FUNCTION_BLOCK SOL_MDL (* Solenoid Model *)
  (* Standard: 61499-1; Classification: Simulation *)
  (* Version 0.1, 2005-06-01, JHC, Holobloc Inc, Recompiled with new emitter. *)
  (* Version 0.0, 2004-09-23, JHC, Rockwell Automation, Simplified, derived from CNV_MDL1. *)
  (* Compiler header: package fb.rt.mva; *)
  (* Compiler Java Sun JDK 1.4.2 *)
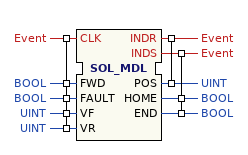
  EVENT_INPUT
    CLK WITH FWD, VF, FAULT, VR; (* Simulation Clock Event *)
  END_EVENT
  EVENT_OUTPUT
    INDR WITH POS; (* Change in Rendering Data *)
    INDS WITH HOME, END; (* Change in Sensor Data *)
  END_EVENT
  VAR_INPUT
    FWD : BOOL; (* Forward motion command *)
    FAULT : BOOL; (* Fault Condition *)
    VF : UINT := 50; (* Forward Speed in % per CLK event *)
    VR : UINT := 50; (* Retract Speed in % per CLK event *)
  END_VAR
  VAR_OUTPUT
    POS : UINT; (* Solenoid Position in % of Conveyor Length *)
    HOME : BOOL; (* Solenoid Fully Retracted *)
    END : BOOL; (* Solenoid Fully Advanced *)
  END_VAR
  ALGORITHM CLK IN Java:
if(FAULT.value) return;
if(FWD.value){
   if(END.value) return;
   if(HOME.value){
      HOME.value = false;
      INDS.serviceEvent(this);}
   POS.value += VF.value;
   if(POS.value >= 100){
      POS.value=100;
      END.value=true;
      INDS.serviceEvent(this);}}
else{
   if (HOME.value) return;
   if(END.value){
      END.value = false;
      INDS.serviceEvent(this);}
   POS.value -= VR.value;
   if(POS.value <= 0){
      POS.value=0;
      HOME.value=true;
      INDS.serviceEvent(this);}}
INDR.serviceEvent(this);
  END_ALGORITHM
END_FUNCTION_BLOCK
